// TwinCAT 3 PLC project RollingAverageTests
// ProgramVersion: 3.1.4026.22
// libraries:
//   Tc2_Standard, * (Beckhoff Automation GmbH)
//   Tc2_System, * (Beckhoff Automation GmbH)
//   TcUnit, * (www.tcunit.org)
//   B1RollingAverage_Plc,newest,Tc3 Project
// project tree:
//   / PlcTask.TcTTO
//   POUs/ FB_RollingAverageConsumer.TcPOU, FB_RollingAverageTests.TcPOU, MAIN.TcPOU
// real-time tasks:
//   TASK PlcTask: cycle T#10ms, priority 20, ADS port 350

CONFIGURATION RollingAverageTests
    RESOURCE PLC ON TwinCAT3
        TASK PlcTask(INTERVAL := T#10ms, PRIORITY := 20);
        PROGRAM MAIN WITH PlcTask : MAIN;
    END_RESOURCE
END_CONFIGURATION

// ---- POUs/MAIN.TcPOU
PROGRAM MAIN
VAR
    suite : FB_RollingAverageTests;
END_VAR

suite();
TcUnit.RUN();

END_PROGRAM

// ---- POUs/FB_RollingAverageTests.TcPOU
FUNCTION_BLOCK FB_RollingAverageTests EXTENDS TcUnit.FB_TestSuite
VAR
    averager : B1RollingAverage_Plc.FB_RollingAverage;
    result : INT;
    i : INT;
END_VAR

AverageOfConstantStream();

METHOD PRIVATE AverageOfConstantStream
TEST('AverageOfConstantStream');
FOR i := 1 TO 8 DO
    result := averager.Step(sample := 10);
END_FOR
AssertEquals_INT(
    Expected := 10,
    Actual := result,
    Message := 'Average of eight 10s should be 10');
TEST_FINISHED();
END_METHOD

END_FUNCTION_BLOCK

// ---- POUs/FB_RollingAverageConsumer.TcPOU
FUNCTION_BLOCK FB_RollingAverageConsumer
VAR
    adder : B1RollingAverage_Plc.FB_RollingAverage;
    lastResult : INT;
END_VAR

lastResult := adder.Step(sample := 10);

END_FUNCTION_BLOCK
